// TIA Portal V15 export
// export: Created 2018-05-29T12:25:38.1552518Z, ExportSetting WithDefaults, DisplayName Totally Integrated Automation Portal, DisplayVersion V15, DisplayName TIA Portal Openness, DisplayVersion V15, DisplayName STEP 7 Professional, DisplayVersion V15, DisplayName WinCC Professional, DisplayVersion V15
FUNCTION "EM_Instance_10_fc" : Void   // FC1, STL
TITLE = _fc
{ S7_Optimized_Access := 'TRUE' }
VERSION : 0.1
// test
// stored: AutoNumber true, UDAEnableTagReadback false
BEGIN

NETWORK
TITLE = Main
// comment:
// Call the EM FB with the corresponding DB instance
CALL EM_I_OUT, EM_Instance_10
	em_id := 35
	Pump_RUN := M106.QNOFF2
	Pump_QERR := M106.QERR
	Pump_EERR := M106.QERR_EXT
	FS01_PV := LS002.QON
	PIC01_PV := FIC101.PV
	PIC01_ERR := FIC101.QERR
	LT01_PV := LT101.QfVal
	LT01_AHH := LT101.LIM_Qb01
	LT01_AH := LT101.LIM_Qb02
	LT01_AL := LT101.LIM_Qb03
	LT01_ALL := LT101.LIM_Qb04
	LT01_ERR := LT101.QERR
	BV_Bottom_OPN := MV007.QOPEN
	BV_Bottom_CLS := MV007.QCLOSE
	BV_Bottom_MERR := MV007.QMON_ERR
	Pump_ON := M106.L_ON
	Pump_AUT := M106.L_AUT
	PIC01_EXT := FIC101.L_REMOTE
	PIC01_SP := FIC101.HMI_SP_INT
	PIC01_AUT := FIC101.L_AUT
	PIC01_VAL_OUT := FIC101.HMI_MAN
	PIC01_SET_SP := FIC101.Set_SP
	PIC01_SET_OUT := FIC101.Set_Output
	BV_Bottom_CMD := MV007.AUT_OP
END_FUNCTION
